PROGRAM PRG_Beamblock
VAR
    fbBEAM_Motor_X : FB_MotionStage;
    fbBEAM_Motor_Y : FB_MotionStage;
    fbBEAM_Motor_Z : FB_MotionStage;
    fbOUTCOUP_Motor_Y : FB_MotionStage;
END_VAR

Main.M30.bHardwareEnable := TRUE;
fbBEAM_Motor_Y(stMotionStage:=Main.M30);

Main.M31.bHardwareEnable := TRUE;
fbBEAM_Motor_X(stMotionStage:=Main.M31);

Main.M32.bHardwareEnable := TRUE;
fbBEAM_Motor_Z(stMotionStage:=Main.M32);

Main.M35.bHardwareEnable := TRUE;
fbOUTCOUP_Motor_Y(stMotionStage:=Main.M35);

END_PROGRAM

(* stored: Version 1.1.0.1, ProductVersion 3.1.4022.18
   POU PRG_Beamblock: Id {cad6a7fa-2f2f-4059-8ecf-4abf4749b17e}, SpecialFunc None *)
